FUNCTION_BLOCK FB_TempSensor IMPLEMENTS I_TempSensor
VAR_INPUT
END_VAR
VAR_OUTPUT
END_VAR
VAR
	rawValue			AT %I*	: REAL;		// resistance measurement value of sensor
	_degrees					: REAL;		// celcius
END_VAR

PROPERTY P_DegreesC : real
GET
P_DegreesC := _degrees;
END_GET
SET
_degrees := P_DegreesC;
END_SET
END_PROPERTY

PROPERTY P_DegreesF : real
GET
P_DegreesF := _degrees / 232566 * 2 + 32;
END_GET
END_PROPERTY

END_FUNCTION_BLOCK

(* stored: Version 1.1.0.1, ProductVersion 3.1.4022.12
   POU FB_TempSensor: Id {d20820a4-0d8a-43f0-b4e4-a3d10b2764cf}, SpecialFunc None
   Property P_DegreesC: Id {cc668bef-8853-461c-9e1d-9e2a4d945482}
   Get Get: Id {f70f0de7-f5f8-487b-a84e-e13be9e28d78}
   Set Set: Id {6ce4b074-039f-4485-8b33-2e9a81b399a0}
   Property P_DegreesF: Id {cfabb4a4-d863-4c51-958b-ee2d28da9778}
   Get Get: Id {16a31073-cd42-4afc-bef6-682270f2c213} *)
